Staubli VAL3: start.pgx

program start()
begin

  clearBuffer(soTcpClient)
  movej(jHome,tGreifer,mUsedSpeed)

  taskCreate "TCP-Server", 10, TCPserver()

  taskCreate "p&p", 5, PickPlace()



  movej(jHome,tGreifer,mUsedSpeed)
  waitEndMove()

end
